FUNCTION_BLOCK BinaryActuator_MDL
  (* Version 1.0, 2005-11-13, Goran Cengic, Chalmers *)
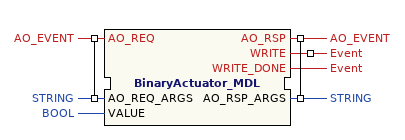
  EVENT_INPUT
    AO_REQ : AO_EVENT WITH AO_REQ_ARGS;
  END_EVENT
  EVENT_OUTPUT
    AO_RSP : AO_EVENT WITH AO_RSP_ARGS;
    WRITE WITH VALUE;
    WRITE_DONE;
  END_EVENT
  VAR_INPUT
    AO_REQ_ARGS : STRING;
    VALUE : BOOL;
  END_VAR
  VAR_OUTPUT
    AO_RSP_ARGS : STRING;
  END_VAR
  VAR
    curValue : BOOL;
  END_VAR
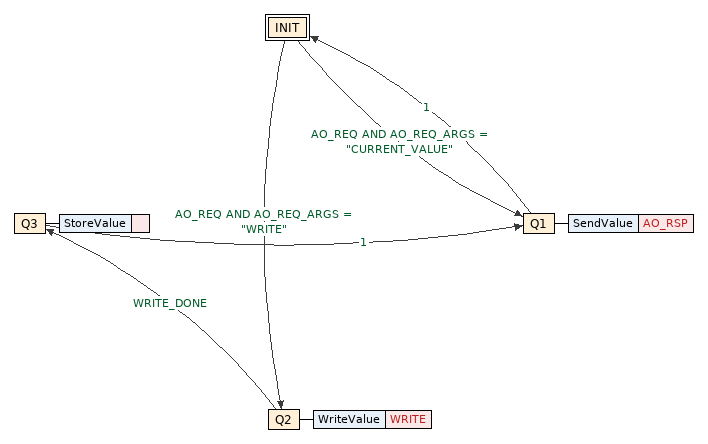
  EC_STATES
    INIT;
    Q1 : SendValue -> AO_RSP;
    Q2 : WriteValue -> WRITE;
    Q3 : StoreValue;
  END_STATES
  EC_TRANSITIONS
    INIT TO Q1 := AO_REQ AND AO_REQ_ARGS = "CURRENT_VALUE";
    Q1 TO INIT := 1;
    INIT TO Q2 := AO_REQ AND AO_REQ_ARGS = "WRITE";
    Q2 TO Q3 := WRITE_DONE;
    Q3 TO Q1 := 1;
  END_TRANSITIONS
  ALGORITHM SendValue IN Java:
AO_RSP_ARGS = "CURRENT_VALUE" + curValue.toString();
  END_ALGORITHM
  ALGORITHM WriteValue IN Java:
VALUE = new Boolean(AO_REQ_ARGS).booleanValue();
  END_ALGORITHM
  ALGORITHM StoreValue IN Java:
curValue = VALUE;
  END_ALGORITHM
END_FUNCTION_BLOCK
